FUNCTION_BLOCK FB_TransportLogik
VAR_INPUT
	bEnable : BOOL;
	bExecute : BOOL;
	eStateE : eBetriebszustand;
	nStation : INT;
	// Logik -> Hardware Signal
	bStation1 : BOOL;
	bStation2 : BOOL;
	bStation3 : BOOL;
	bStation4 : BOOL;
END_VAR
VAR_OUTPUT
	bEnableA : BOOL;
	bExecuteA : BOOL;
	bStopA : BOOL;
	eStateA: eBetriebszustand;
	bStop1 : BOOL;
	bStop2 : BOOL;
	bStop3 : BOOL;
END_VAR
VAR
	nState : INT;
END_VAR

END_FUNCTION_BLOCK

(* stored: Version 1.1.0.1, ProductVersion 3.1.4024.15
   POU FB_TransportLogik: Id {024fb3a1-fd5b-4664-9520-3d063823ae19}, SpecialFunc None *)
